FUNCTION_BLOCK ADS_SERVER_CONFIG (* Service Interface Function Block Type *)
  (* Standard: 61499-2; Description: Copyright (c) 2018 TU Vienna/ACIN This program and the accompanying materials are made available under the terms of the Eclipse Public License 2.0 which is available at https://www.eclipse.org/legal/epl-2.0/ SPDX-License-Identifier: EPL-2.0 *)
  (* Version 1.0, 2018-08-28, Martin Melik Merkumians, TU Vienna/ACIN *)
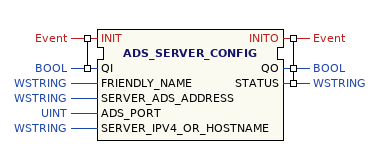
  EVENT_INPUT
    INIT WITH QI; (* Service Initialization *)
  END_EVENT
  EVENT_OUTPUT
    INITO WITH QO, STATUS; (* Initialization Confirm *)
  END_EVENT
  VAR_INPUT
    QI : BOOL; (* Event Input Qualifier *)
    FRIENDLY_NAME : WSTRING; (* User friendly server name to use in IO FBs *)
    SERVER_ADS_ADDRESS : WSTRING; (* Server ADS address *)
    ADS_PORT : UINT; (* Server ADS port *)
    SERVER_IPV4_OR_HOSTNAME : WSTRING; (* ADS Server IPv4 address or hostame *)
  END_VAR
  VAR_OUTPUT
    QO : BOOL; (* Event Output Qualifier *)
    STATUS : WSTRING; (* Service Status *)
  END_VAR
END_FUNCTION_BLOCK
